TYPE "UDT_ZC_CONTADOR_MINUTOS"
TITLE = ZC_CONTADOR_MINUTOS
VERSION : 0.1
//Tipo de dato contador tiempo
   STRUCT
      Minuto : UDInt;   // Contador Minutos
      Segundo : USInt;   // Contador Segundos
   END_STRUCT;

END_TYPE

